Staubli VAL3: start.pgx

public program start()
begin
  // Program Rect10 start
  // Program generated by RoboDK v3.6.2 for Staubli TX200 on 17/05/2019 09:38:33
  // Using nominal kinematics.
   // mise en rotation pompe vitesse nulle
   aioSet(Tpompe,0)
   put("Tension pompe nulle")
   // arrêt pompe
   dioSet(doPompe,0)
   put("Pompe arret")

   // fermeture obturateur
   dioSet(doValve2,0)
   dioSet(doValve1,1)
   put("Obturateur fermé")
  // Afficher effecteur
  nTraj=movej(jJoint[0],tTool[0],mSpeed[0])
  nTraj=movel(pPoint[0],tTool[0],mSpeed[0])
  nTraj=movel(pPoint[1],tTool[0],mSpeed[0])
  waitEndMove()

  // ouverture obturateur
  dioSet(doValve1,0)
  dioSet(doValve2,1)
  put("Obturateur ouvert")
  delay(nTObtOpen)
  // marche pompe vitesse faible
  dioSet(doPompe,1)
  put("Pompe en marche")
  delay(nTPompeOn)
  // rotation pompe vitesse donnée
  aioSet(Tpompe,nTension)
  put("Pompe en rotation")
  nTraj=movel(pPoint[2],tTool[0],mSpeed[0])
  nTraj=movel(pPoint[3],tTool[0],mSpeed[1])
  nTraj=movel(pPoint[4],tTool[0],mSpeed[1])
  nTraj=movel(pPoint[5],tTool[0],mSpeed[1])
  nTraj=movel(pPoint[6],tTool[0],mSpeed[1])
  nTraj=movel(pPoint[7],tTool[0],mSpeed[1])
  nTraj=movel(pPoint[8],tTool[0],mSpeed[1])
  nTraj=movel(pPoint[9],tTool[0],mSpeed[1])
  nTraj=movel(pPoint[10],tTool[0],mSpeed[1])
  nTraj=movel(pPoint[11],tTool[0],mSpeed[1])
  nTraj=movel(pPoint[12],tTool[0],mSpeed[1])
  nTraj=movel(pPoint[13],tTool[0],mSpeed[1])
  nTraj=movel(pPoint[14],tTool[0],mSpeed[1])
  nTraj=movel(pPoint[15],tTool[0],mSpeed[1])
  nTraj=movel(pPoint[16],tTool[0],mSpeed[1])
  nTraj=movel(pPoint[17],tTool[0],mSpeed[1])
  nTraj=movel(pPoint[18],tTool[0],mSpeed[1])
  nTraj=movel(pPoint[19],tTool[0],mSpeed[1])
  nTraj=movel(pPoint[20],tTool[0],mSpeed[1])
  nTraj=movel(pPoint[21],tTool[0],mSpeed[1])
  nTraj=movel(pPoint[22],tTool[0],mSpeed[1])
  nTraj=movel(pPoint[23],tTool[0],mSpeed[1])
  nTraj=movel(pPoint[24],tTool[0],mSpeed[1])
  nTraj=movel(pPoint[25],tTool[0],mSpeed[1])
  nTraj=movel(pPoint[26],tTool[0],mSpeed[1])
  nTraj=movel(pPoint[27],tTool[0],mSpeed[1])
  nTraj=movel(pPoint[28],tTool[0],mSpeed[1])
  nTraj=movel(pPoint[29],tTool[0],mSpeed[1])
  nTraj=movel(pPoint[30],tTool[0],mSpeed[1])
  nTraj=movel(pPoint[31],tTool[0],mSpeed[1])
  nTraj=movel(pPoint[32],tTool[0],mSpeed[1])
  nTraj=movel(pPoint[33],tTool[0],mSpeed[1])
  nTraj=movel(pPoint[34],tTool[0],mSpeed[1])
  nTraj=movel(pPoint[35],tTool[0],mSpeed[1])
  nTraj=movel(pPoint[36],tTool[0],mSpeed[1])
  nTraj=movel(pPoint[37],tTool[0],mSpeed[1])
  nTraj=movel(pPoint[38],tTool[0],mSpeed[1])
  nTraj=movel(pPoint[39],tTool[0],mSpeed[1])
  nTraj=movel(pPoint[40],tTool[0],mSpeed[1])
  nTraj=movel(pPoint[41],tTool[0],mSpeed[1])
  nTraj=movel(pPoint[42],tTool[0],mSpeed[1])
  nTraj=movel(pPoint[43],tTool[0],mSpeed[1])
  nTraj=movel(pPoint[44],tTool[0],mSpeed[1])
  nTraj=movel(pPoint[45],tTool[0],mSpeed[1])
  nTraj=movel(pPoint[46],tTool[0],mSpeed[1])
  nTraj=movel(pPoint[47],tTool[0],mSpeed[1])
  nTraj=movel(pPoint[48],tTool[0],mSpeed[1])
  nTraj=movel(pPoint[49],tTool[0],mSpeed[1])
  nTraj=movel(pPoint[50],tTool[0],mSpeed[1])
  nTraj=movel(pPoint[51],tTool[0],mSpeed[1])
  nTraj=movel(pPoint[52],tTool[0],mSpeed[1])
  nTraj=movel(pPoint[53],tTool[0],mSpeed[1])
  nTraj=movel(pPoint[54],tTool[0],mSpeed[1])
  nTraj=movel(pPoint[55],tTool[0],mSpeed[1])
  nTraj=movel(pPoint[56],tTool[0],mSpeed[1])
  nTraj=movel(pPoint[57],tTool[0],mSpeed[1])
  nTraj=movel(pPoint[58],tTool[0],mSpeed[1])
  nTraj=movel(pPoint[59],tTool[0],mSpeed[1])
  nTraj=movel(pPoint[60],tTool[0],mSpeed[1])
  nTraj=movel(pPoint[61],tTool[0],mSpeed[1])
  nTraj=movel(pPoint[62],tTool[0],mSpeed[1])
  nTraj=movel(pPoint[63],tTool[0],mSpeed[1])
  nTraj=movel(pPoint[64],tTool[0],mSpeed[1])
  nTraj=movel(pPoint[65],tTool[0],mSpeed[1])
  nTraj=movel(pPoint[66],tTool[0],mSpeed[1])
  nTraj=movel(pPoint[67],tTool[0],mSpeed[1])
  nTraj=movel(pPoint[68],tTool[0],mSpeed[1])
  nTraj=movel(pPoint[69],tTool[0],mSpeed[1])
  nTraj=movel(pPoint[70],tTool[0],mSpeed[1])
  waitEndMove()
    // arrêt pompe
  dioSet(doPompe,0)
  put("Pompe arret")
  delay(nTPompeOff)

  // fermeture obturateur
  dioSet(doValve2,0)
  dioSet(doValve1,1)
  put("Obturateur fermé")
  nTraj=movel(pPoint[71],tTool[0],mSpeed[1])
  waitEndMove()

  nTraj=movel(pPoint[72],tTool[0],mSpeed[2])
  nTraj=movel(pPoint[73],tTool[0],mSpeed[2])
  nTraj=movel(pPoint[74],tTool[0],mSpeed[3])
  nTraj=movel(pPoint[75],tTool[0],mSpeed[3])
  waitEndMove()

  // ouverture obturateur
  dioSet(doValve1,0)
  dioSet(doValve2,1)
  put("Obturateur ouvert")
  delay(nTObtOpen)
  // marche pompe vitesse faible
  dioSet(doPompe,1)
  put("Pompe en marche")
  delay(nTPompeOn)
  // rotation pompe vitesse donnée
  aioSet(Tpompe,nTension)
  put("Pompe en rotation")
  nTraj=movel(pPoint[76],tTool[0],mSpeed[3])
  nTraj=movel(pPoint[77],tTool[0],mSpeed[4])
  nTraj=movel(pPoint[78],tTool[0],mSpeed[4])
  nTraj=movel(pPoint[79],tTool[0],mSpeed[4])
  nTraj=movel(pPoint[80],tTool[0],mSpeed[4])
  nTraj=movel(pPoint[81],tTool[0],mSpeed[4])
  nTraj=movel(pPoint[82],tTool[0],mSpeed[4])
  nTraj=movel(pPoint[83],tTool[0],mSpeed[4])
  nTraj=movel(pPoint[84],tTool[0],mSpeed[4])
  nTraj=movel(pPoint[85],tTool[0],mSpeed[4])
  nTraj=movel(pPoint[86],tTool[0],mSpeed[4])
  nTraj=movel(pPoint[87],tTool[0],mSpeed[4])
  nTraj=movel(pPoint[88],tTool[0],mSpeed[4])
  nTraj=movel(pPoint[89],tTool[0],mSpeed[4])
  nTraj=movel(pPoint[90],tTool[0],mSpeed[4])
  nTraj=movel(pPoint[91],tTool[0],mSpeed[4])
  nTraj=movel(pPoint[92],tTool[0],mSpeed[4])
  nTraj=movel(pPoint[93],tTool[0],mSpeed[4])
  nTraj=movel(pPoint[94],tTool[0],mSpeed[4])
  nTraj=movel(pPoint[95],tTool[0],mSpeed[4])
  nTraj=movel(pPoint[96],tTool[0],mSpeed[4])
  nTraj=movel(pPoint[97],tTool[0],mSpeed[4])
  nTraj=movel(pPoint[98],tTool[0],mSpeed[4])
  nTraj=movel(pPoint[99],tTool[0],mSpeed[4])
  nTraj=movel(pPoint[100],tTool[0],mSpeed[4])
  nTraj=movel(pPoint[101],tTool[0],mSpeed[4])
  nTraj=movel(pPoint[102],tTool[0],mSpeed[4])
  nTraj=movel(pPoint[103],tTool[0],mSpeed[4])
  nTraj=movel(pPoint[104],tTool[0],mSpeed[4])
  nTraj=movel(pPoint[105],tTool[0],mSpeed[4])
  nTraj=movel(pPoint[106],tTool[0],mSpeed[4])
  nTraj=movel(pPoint[107],tTool[0],mSpeed[4])
  nTraj=movel(pPoint[108],tTool[0],mSpeed[4])
  nTraj=movel(pPoint[109],tTool[0],mSpeed[4])
  nTraj=movel(pPoint[110],tTool[0],mSpeed[4])
  nTraj=movel(pPoint[111],tTool[0],mSpeed[4])
  nTraj=movel(pPoint[112],tTool[0],mSpeed[4])
  nTraj=movel(pPoint[113],tTool[0],mSpeed[4])
  nTraj=movel(pPoint[114],tTool[0],mSpeed[4])
  nTraj=movel(pPoint[115],tTool[0],mSpeed[4])
  nTraj=movel(pPoint[116],tTool[0],mSpeed[4])
  nTraj=movel(pPoint[117],tTool[0],mSpeed[4])
  nTraj=movel(pPoint[118],tTool[0],mSpeed[4])
  nTraj=movel(pPoint[119],tTool[0],mSpeed[4])
  nTraj=movel(pPoint[120],tTool[0],mSpeed[4])
  nTraj=movel(pPoint[121],tTool[0],mSpeed[4])
  nTraj=movel(pPoint[122],tTool[0],mSpeed[4])
  nTraj=movel(pPoint[123],tTool[0],mSpeed[4])
  nTraj=movel(pPoint[124],tTool[0],mSpeed[4])
  nTraj=movel(pPoint[125],tTool[0],mSpeed[4])
  nTraj=movel(pPoint[126],tTool[0],mSpeed[4])
  nTraj=movel(pPoint[127],tTool[0],mSpeed[4])
  nTraj=movel(pPoint[128],tTool[0],mSpeed[4])
  nTraj=movel(pPoint[129],tTool[0],mSpeed[4])
  nTraj=movel(pPoint[130],tTool[0],mSpeed[4])
  nTraj=movel(pPoint[131],tTool[0],mSpeed[4])
  nTraj=movel(pPoint[132],tTool[0],mSpeed[4])
  nTraj=movel(pPoint[133],tTool[0],mSpeed[4])
  nTraj=movel(pPoint[134],tTool[0],mSpeed[4])
  nTraj=movel(pPoint[135],tTool[0],mSpeed[4])
  nTraj=movel(pPoint[136],tTool[0],mSpeed[4])
  nTraj=movel(pPoint[137],tTool[0],mSpeed[4])
  nTraj=movel(pPoint[138],tTool[0],mSpeed[4])
  nTraj=movel(pPoint[139],tTool[0],mSpeed[4])
  nTraj=movel(pPoint[140],tTool[0],mSpeed[4])
  nTraj=movel(pPoint[141],tTool[0],mSpeed[4])
  nTraj=movel(pPoint[142],tTool[0],mSpeed[4])
  nTraj=movel(pPoint[143],tTool[0],mSpeed[4])
  nTraj=movel(pPoint[144],tTool[0],mSpeed[4])
    waitEndMove()

  // arrêt pompe
  dioSet(doPompe,0)
  put("Pompe arret")
  delay(nTPompeOff)

  // fermeture obturateur
  dioSet(doValve2,0)
  dioSet(doValve1,1)
  put("Obturateur fermé")
  nTraj=movel(pPoint[145],tTool[0],mSpeed[4])
  waitEndMove()

  nTraj=movel(pPoint[146],tTool[0],mSpeed[5])
  nTraj=movel(pPoint[147],tTool[0],mSpeed[5])
  nTraj=movel(pPoint[148],tTool[0],mSpeed[6])
  nTraj=movel(pPoint[149],tTool[0],mSpeed[6])
  waitEndMove()

  // ouverture obturateur
  dioSet(doValve1,0)
  dioSet(doValve2,1)
  put("Obturateur ouvert")
  delay(nTObtOpen)
  // marche pompe vitesse faible
  dioSet(doPompe,1)
  put("Pompe en marche")
  delay(nTPompeOn)
  // rotation pompe vitesse donnée
  aioSet(Tpompe,nTension)
  put("Pompe en rotation")
  nTraj=movel(pPoint[150],tTool[0],mSpeed[6])
  nTraj=movel(pPoint[151],tTool[0],mSpeed[7])
  nTraj=movel(pPoint[152],tTool[0],mSpeed[7])
  nTraj=movel(pPoint[153],tTool[0],mSpeed[7])
  nTraj=movel(pPoint[154],tTool[0],mSpeed[7])
  nTraj=movel(pPoint[155],tTool[0],mSpeed[7])
  nTraj=movel(pPoint[156],tTool[0],mSpeed[7])
  nTraj=movel(pPoint[157],tTool[0],mSpeed[7])
  nTraj=movel(pPoint[158],tTool[0],mSpeed[7])
  nTraj=movel(pPoint[159],tTool[0],mSpeed[7])
  nTraj=movel(pPoint[160],tTool[0],mSpeed[7])
  nTraj=movel(pPoint[161],tTool[0],mSpeed[7])
  nTraj=movel(pPoint[162],tTool[0],mSpeed[7])
  nTraj=movel(pPoint[163],tTool[0],mSpeed[7])
  nTraj=movel(pPoint[164],tTool[0],mSpeed[7])
  nTraj=movel(pPoint[165],tTool[0],mSpeed[7])
  nTraj=movel(pPoint[166],tTool[0],mSpeed[7])
  nTraj=movel(pPoint[167],tTool[0],mSpeed[7])
  nTraj=movel(pPoint[168],tTool[0],mSpeed[7])
  nTraj=movel(pPoint[169],tTool[0],mSpeed[7])
  nTraj=movel(pPoint[170],tTool[0],mSpeed[7])
  nTraj=movel(pPoint[171],tTool[0],mSpeed[7])
  nTraj=movel(pPoint[172],tTool[0],mSpeed[7])
  nTraj=movel(pPoint[173],tTool[0],mSpeed[7])
  nTraj=movel(pPoint[174],tTool[0],mSpeed[7])
  nTraj=movel(pPoint[175],tTool[0],mSpeed[7])
  nTraj=movel(pPoint[176],tTool[0],mSpeed[7])
  nTraj=movel(pPoint[177],tTool[0],mSpeed[7])
  nTraj=movel(pPoint[178],tTool[0],mSpeed[7])
  nTraj=movel(pPoint[179],tTool[0],mSpeed[7])
  nTraj=movel(pPoint[180],tTool[0],mSpeed[7])
  nTraj=movel(pPoint[181],tTool[0],mSpeed[7])
  nTraj=movel(pPoint[182],tTool[0],mSpeed[7])
  nTraj=movel(pPoint[183],tTool[0],mSpeed[7])
  nTraj=movel(pPoint[184],tTool[0],mSpeed[7])
  nTraj=movel(pPoint[185],tTool[0],mSpeed[7])
  nTraj=movel(pPoint[186],tTool[0],mSpeed[7])
  nTraj=movel(pPoint[187],tTool[0],mSpeed[7])
  nTraj=movel(pPoint[188],tTool[0],mSpeed[7])
  nTraj=movel(pPoint[189],tTool[0],mSpeed[7])
  nTraj=movel(pPoint[190],tTool[0],mSpeed[7])
  nTraj=movel(pPoint[191],tTool[0],mSpeed[7])
  nTraj=movel(pPoint[192],tTool[0],mSpeed[7])
  nTraj=movel(pPoint[193],tTool[0],mSpeed[7])
  nTraj=movel(pPoint[194],tTool[0],mSpeed[7])
  nTraj=movel(pPoint[195],tTool[0],mSpeed[7])
  nTraj=movel(pPoint[196],tTool[0],mSpeed[7])
  nTraj=movel(pPoint[197],tTool[0],mSpeed[7])
  nTraj=movel(pPoint[198],tTool[0],mSpeed[7])
  nTraj=movel(pPoint[199],tTool[0],mSpeed[7])
  nTraj=movel(pPoint[200],tTool[0],mSpeed[7])
  nTraj=movel(pPoint[201],tTool[0],mSpeed[7])
  nTraj=movel(pPoint[202],tTool[0],mSpeed[7])
  nTraj=movel(pPoint[203],tTool[0],mSpeed[7])
  nTraj=movel(pPoint[204],tTool[0],mSpeed[7])
  nTraj=movel(pPoint[205],tTool[0],mSpeed[7])
  nTraj=movel(pPoint[206],tTool[0],mSpeed[7])
  nTraj=movel(pPoint[207],tTool[0],mSpeed[7])
  nTraj=movel(pPoint[208],tTool[0],mSpeed[7])
  nTraj=movel(pPoint[209],tTool[0],mSpeed[7])
  nTraj=movel(pPoint[210],tTool[0],mSpeed[7])
  nTraj=movel(pPoint[211],tTool[0],mSpeed[7])
  nTraj=movel(pPoint[212],tTool[0],mSpeed[7])
  nTraj=movel(pPoint[213],tTool[0],mSpeed[7])
  nTraj=movel(pPoint[214],tTool[0],mSpeed[7])
  nTraj=movel(pPoint[215],tTool[0],mSpeed[7])
  nTraj=movel(pPoint[216],tTool[0],mSpeed[7])
  nTraj=movel(pPoint[217],tTool[0],mSpeed[7])
  nTraj=movel(pPoint[218],tTool[0],mSpeed[7])
    waitEndMove()

  // arrêt pompe
  dioSet(doPompe,0)
  put("Pompe arret")
  delay(nTPompeOff)

  // fermeture obturateur
  dioSet(doValve2,0)
  dioSet(doValve1,1)
  put("Obturateur fermé")
  nTraj=movel(pPoint[219],tTool[0],mSpeed[7])
  waitEndMove()

  nTraj=movel(pPoint[220],tTool[0],mSpeed[8])
  nTraj=movel(pPoint[221],tTool[0],mSpeed[8])
  nTraj=movel(pPoint[222],tTool[0],mSpeed[9])
  nTraj=movel(pPoint[223],tTool[0],mSpeed[9])
  waitEndMove()

  // ouverture obturateur
  dioSet(doValve1,0)
  dioSet(doValve2,1)
  put("Obturateur ouvert")
  delay(nTObtOpen)
  // marche pompe vitesse faible
  dioSet(doPompe,1)
  put("Pompe en marche")
  delay(nTPompeOn)
  // rotation pompe vitesse donnée
  aioSet(Tpompe,nTension)
  put("Pompe en rotation")
  nTraj=movel(pPoint[224],tTool[0],mSpeed[9])
  nTraj=movel(pPoint[225],tTool[0],mSpeed[10])
  nTraj=movel(pPoint[226],tTool[0],mSpeed[10])
  nTraj=movel(pPoint[227],tTool[0],mSpeed[10])
  nTraj=movel(pPoint[228],tTool[0],mSpeed[10])
  nTraj=movel(pPoint[229],tTool[0],mSpeed[10])
  nTraj=movel(pPoint[230],tTool[0],mSpeed[10])
  nTraj=movel(pPoint[231],tTool[0],mSpeed[10])
  nTraj=movel(pPoint[232],tTool[0],mSpeed[10])
  nTraj=movel(pPoint[233],tTool[0],mSpeed[10])
  nTraj=movel(pPoint[234],tTool[0],mSpeed[10])
  nTraj=movel(pPoint[235],tTool[0],mSpeed[10])
  nTraj=movel(pPoint[236],tTool[0],mSpeed[10])
  nTraj=movel(pPoint[237],tTool[0],mSpeed[10])
  nTraj=movel(pPoint[238],tTool[0],mSpeed[10])
  nTraj=movel(pPoint[239],tTool[0],mSpeed[10])
  nTraj=movel(pPoint[240],tTool[0],mSpeed[10])
  nTraj=movel(pPoint[241],tTool[0],mSpeed[10])
  nTraj=movel(pPoint[242],tTool[0],mSpeed[10])
  nTraj=movel(pPoint[243],tTool[0],mSpeed[10])
  nTraj=movel(pPoint[244],tTool[0],mSpeed[10])
  nTraj=movel(pPoint[245],tTool[0],mSpeed[10])
  nTraj=movel(pPoint[246],tTool[0],mSpeed[10])
  nTraj=movel(pPoint[247],tTool[0],mSpeed[10])
  nTraj=movel(pPoint[248],tTool[0],mSpeed[10])
  nTraj=movel(pPoint[249],tTool[0],mSpeed[10])
  nTraj=movel(pPoint[250],tTool[0],mSpeed[10])
  nTraj=movel(pPoint[251],tTool[0],mSpeed[10])
  nTraj=movel(pPoint[252],tTool[0],mSpeed[10])
  nTraj=movel(pPoint[253],tTool[0],mSpeed[10])
  nTraj=movel(pPoint[254],tTool[0],mSpeed[10])
  nTraj=movel(pPoint[255],tTool[0],mSpeed[10])
  nTraj=movel(pPoint[256],tTool[0],mSpeed[10])
  nTraj=movel(pPoint[257],tTool[0],mSpeed[10])
  nTraj=movel(pPoint[258],tTool[0],mSpeed[10])
  nTraj=movel(pPoint[259],tTool[0],mSpeed[10])
  nTraj=movel(pPoint[260],tTool[0],mSpeed[10])
  nTraj=movel(pPoint[261],tTool[0],mSpeed[10])
  nTraj=movel(pPoint[262],tTool[0],mSpeed[10])
  nTraj=movel(pPoint[263],tTool[0],mSpeed[10])
  nTraj=movel(pPoint[264],tTool[0],mSpeed[10])
  nTraj=movel(pPoint[265],tTool[0],mSpeed[10])
  nTraj=movel(pPoint[266],tTool[0],mSpeed[10])
  nTraj=movel(pPoint[267],tTool[0],mSpeed[10])
  nTraj=movel(pPoint[268],tTool[0],mSpeed[10])
  nTraj=movel(pPoint[269],tTool[0],mSpeed[10])
  nTraj=movel(pPoint[270],tTool[0],mSpeed[10])
  nTraj=movel(pPoint[271],tTool[0],mSpeed[10])
  nTraj=movel(pPoint[272],tTool[0],mSpeed[10])
  nTraj=movel(pPoint[273],tTool[0],mSpeed[10])
  nTraj=movel(pPoint[274],tTool[0],mSpeed[10])
  nTraj=movel(pPoint[275],tTool[0],mSpeed[10])
  nTraj=movel(pPoint[276],tTool[0],mSpeed[10])
  nTraj=movel(pPoint[277],tTool[0],mSpeed[10])
  nTraj=movel(pPoint[278],tTool[0],mSpeed[10])
  nTraj=movel(pPoint[279],tTool[0],mSpeed[10])
  nTraj=movel(pPoint[280],tTool[0],mSpeed[10])
  nTraj=movel(pPoint[281],tTool[0],mSpeed[10])
  nTraj=movel(pPoint[282],tTool[0],mSpeed[10])
  nTraj=movel(pPoint[283],tTool[0],mSpeed[10])
  nTraj=movel(pPoint[284],tTool[0],mSpeed[10])
  nTraj=movel(pPoint[285],tTool[0],mSpeed[10])
  nTraj=movel(pPoint[286],tTool[0],mSpeed[10])
  nTraj=movel(pPoint[287],tTool[0],mSpeed[10])
  nTraj=movel(pPoint[288],tTool[0],mSpeed[10])
  nTraj=movel(pPoint[289],tTool[0],mSpeed[10])
  nTraj=movel(pPoint[290],tTool[0],mSpeed[10])
  nTraj=movel(pPoint[291],tTool[0],mSpeed[10])
  nTraj=movel(pPoint[292],tTool[0],mSpeed[10])
    waitEndMove()

  // arrêt pompe
  dioSet(doPompe,0)
  put("Pompe arret")
  delay(nTPompeOff)

  // fermeture obturateur
  dioSet(doValve2,0)
  dioSet(doValve1,1)
  put("Obturateur fermé")
  nTraj=movel(pPoint[293],tTool[0],mSpeed[10])
  waitEndMove()


  nTraj=movel(pPoint[294],tTool[0],mSpeed[11])
  nTraj=movel(pPoint[295],tTool[0],mSpeed[11])
  nTraj=movel(pPoint[296],tTool[0],mSpeed[12])
  nTraj=movel(pPoint[297],tTool[0],mSpeed[12])
  waitEndMove()

  // ouverture obturateur
  dioSet(doValve1,0)
  dioSet(doValve2,1)
  put("Obturateur ouvert")
  delay(nTObtOpen)
  // marche pompe vitesse faible
  dioSet(doPompe,1)
  put("Pompe en marche")
  delay(nTPompeOn)
  // rotation pompe vitesse donnée
  aioSet(Tpompe,nTension)
  put("Pompe en rotation")
  nTraj=movel(pPoint[298],tTool[0],mSpeed[12])
  nTraj=movel(pPoint[299],tTool[0],mSpeed[13])
  nTraj=movel(pPoint[300],tTool[0],mSpeed[13])
  nTraj=movel(pPoint[301],tTool[0],mSpeed[13])
  nTraj=movel(pPoint[302],tTool[0],mSpeed[13])
  nTraj=movel(pPoint[303],tTool[0],mSpeed[13])
  nTraj=movel(pPoint[304],tTool[0],mSpeed[13])
  nTraj=movel(pPoint[305],tTool[0],mSpeed[13])
  nTraj=movel(pPoint[306],tTool[0],mSpeed[13])
  nTraj=movel(pPoint[307],tTool[0],mSpeed[13])
  nTraj=movel(pPoint[308],tTool[0],mSpeed[13])
  nTraj=movel(pPoint[309],tTool[0],mSpeed[13])
  nTraj=movel(pPoint[310],tTool[0],mSpeed[13])
  nTraj=movel(pPoint[311],tTool[0],mSpeed[13])
  nTraj=movel(pPoint[312],tTool[0],mSpeed[13])
  nTraj=movel(pPoint[313],tTool[0],mSpeed[13])
  nTraj=movel(pPoint[314],tTool[0],mSpeed[13])
  nTraj=movel(pPoint[315],tTool[0],mSpeed[13])
  nTraj=movel(pPoint[316],tTool[0],mSpeed[13])
  nTraj=movel(pPoint[317],tTool[0],mSpeed[13])
  nTraj=movel(pPoint[318],tTool[0],mSpeed[13])
  nTraj=movel(pPoint[319],tTool[0],mSpeed[13])
  nTraj=movel(pPoint[320],tTool[0],mSpeed[13])
  nTraj=movel(pPoint[321],tTool[0],mSpeed[13])
  nTraj=movel(pPoint[322],tTool[0],mSpeed[13])
  nTraj=movel(pPoint[323],tTool[0],mSpeed[13])
  nTraj=movel(pPoint[324],tTool[0],mSpeed[13])
  nTraj=movel(pPoint[325],tTool[0],mSpeed[13])
  nTraj=movel(pPoint[326],tTool[0],mSpeed[13])
  nTraj=movel(pPoint[327],tTool[0],mSpeed[13])
  nTraj=movel(pPoint[328],tTool[0],mSpeed[13])
  nTraj=movel(pPoint[329],tTool[0],mSpeed[13])
  nTraj=movel(pPoint[330],tTool[0],mSpeed[13])
  nTraj=movel(pPoint[331],tTool[0],mSpeed[13])
  nTraj=movel(pPoint[332],tTool[0],mSpeed[13])
  nTraj=movel(pPoint[333],tTool[0],mSpeed[13])
  nTraj=movel(pPoint[334],tTool[0],mSpeed[13])
  nTraj=movel(pPoint[335],tTool[0],mSpeed[13])
  nTraj=movel(pPoint[336],tTool[0],mSpeed[13])
  nTraj=movel(pPoint[337],tTool[0],mSpeed[13])
  nTraj=movel(pPoint[338],tTool[0],mSpeed[13])
  nTraj=movel(pPoint[339],tTool[0],mSpeed[13])
  nTraj=movel(pPoint[340],tTool[0],mSpeed[13])
  nTraj=movel(pPoint[341],tTool[0],mSpeed[13])
  nTraj=movel(pPoint[342],tTool[0],mSpeed[13])
  nTraj=movel(pPoint[343],tTool[0],mSpeed[13])
  nTraj=movel(pPoint[344],tTool[0],mSpeed[13])
  nTraj=movel(pPoint[345],tTool[0],mSpeed[13])
  nTraj=movel(pPoint[346],tTool[0],mSpeed[13])
  nTraj=movel(pPoint[347],tTool[0],mSpeed[13])
  nTraj=movel(pPoint[348],tTool[0],mSpeed[13])
  nTraj=movel(pPoint[349],tTool[0],mSpeed[13])
  nTraj=movel(pPoint[350],tTool[0],mSpeed[13])
  nTraj=movel(pPoint[351],tTool[0],mSpeed[13])
  nTraj=movel(pPoint[352],tTool[0],mSpeed[13])
  nTraj=movel(pPoint[353],tTool[0],mSpeed[13])
  nTraj=movel(pPoint[354],tTool[0],mSpeed[13])
  nTraj=movel(pPoint[355],tTool[0],mSpeed[13])
  nTraj=movel(pPoint[356],tTool[0],mSpeed[13])
  nTraj=movel(pPoint[357],tTool[0],mSpeed[13])
  nTraj=movel(pPoint[358],tTool[0],mSpeed[13])
  nTraj=movel(pPoint[359],tTool[0],mSpeed[13])
  nTraj=movel(pPoint[360],tTool[0],mSpeed[13])
  nTraj=movel(pPoint[361],tTool[0],mSpeed[13])
  nTraj=movel(pPoint[362],tTool[0],mSpeed[13])
  nTraj=movel(pPoint[363],tTool[0],mSpeed[13])
  nTraj=movel(pPoint[364],tTool[0],mSpeed[13])
  nTraj=movel(pPoint[365],tTool[0],mSpeed[13])
  nTraj=movel(pPoint[366],tTool[0],mSpeed[13])
    waitEndMove()

  // arrêt pompe
  dioSet(doPompe,0)
  put("Pompe arret")
  delay(nTPompeOff)

  // fermeture obturateur
  dioSet(doValve2,0)
  dioSet(doValve1,1)
  put("Obturateur fermé")
  nTraj=movel(pPoint[367],tTool[0],mSpeed[13])
  waitEndMove()

  nTraj=movel(pPoint[368],tTool[0],mSpeed[14])
  nTraj=movel(pPoint[369],tTool[0],mSpeed[14])
  nTraj=movel(pPoint[370],tTool[0],mSpeed[15])
  nTraj=movel(pPoint[371],tTool[0],mSpeed[15])
  waitEndMove()

  // ouverture obturateur
  dioSet(doValve1,0)
  dioSet(doValve2,1)
  put("Obturateur ouvert")
  delay(nTObtOpen)
  // marche pompe vitesse faible
  dioSet(doPompe,1)
  put("Pompe en marche")
  delay(nTPompeOn)
  // rotation pompe vitesse donnée
  aioSet(Tpompe,nTension)
  put("Pompe en rotation")
  nTraj=movel(pPoint[372],tTool[0],mSpeed[15])
  nTraj=movel(pPoint[373],tTool[0],mSpeed[16])
  nTraj=movel(pPoint[374],tTool[0],mSpeed[16])
  nTraj=movel(pPoint[375],tTool[0],mSpeed[16])
  nTraj=movel(pPoint[376],tTool[0],mSpeed[16])
  nTraj=movel(pPoint[377],tTool[0],mSpeed[16])
  nTraj=movel(pPoint[378],tTool[0],mSpeed[16])
  nTraj=movel(pPoint[379],tTool[0],mSpeed[16])
  nTraj=movel(pPoint[380],tTool[0],mSpeed[16])
  nTraj=movel(pPoint[381],tTool[0],mSpeed[16])
  nTraj=movel(pPoint[382],tTool[0],mSpeed[16])
  nTraj=movel(pPoint[383],tTool[0],mSpeed[16])
  nTraj=movel(pPoint[384],tTool[0],mSpeed[16])
  nTraj=movel(pPoint[385],tTool[0],mSpeed[16])
  nTraj=movel(pPoint[386],tTool[0],mSpeed[16])
  nTraj=movel(pPoint[387],tTool[0],mSpeed[16])
  nTraj=movel(pPoint[388],tTool[0],mSpeed[16])
  nTraj=movel(pPoint[389],tTool[0],mSpeed[16])
  nTraj=movel(pPoint[390],tTool[0],mSpeed[16])
  nTraj=movel(pPoint[391],tTool[0],mSpeed[16])
  nTraj=movel(pPoint[392],tTool[0],mSpeed[16])
  nTraj=movel(pPoint[393],tTool[0],mSpeed[16])
  nTraj=movel(pPoint[394],tTool[0],mSpeed[16])
  nTraj=movel(pPoint[395],tTool[0],mSpeed[16])
  nTraj=movel(pPoint[396],tTool[0],mSpeed[16])
  nTraj=movel(pPoint[397],tTool[0],mSpeed[16])
  nTraj=movel(pPoint[398],tTool[0],mSpeed[16])
  nTraj=movel(pPoint[399],tTool[0],mSpeed[16])
  nTraj=movel(pPoint[400],tTool[0],mSpeed[16])
  nTraj=movel(pPoint[401],tTool[0],mSpeed[16])
  nTraj=movel(pPoint[402],tTool[0],mSpeed[16])
  nTraj=movel(pPoint[403],tTool[0],mSpeed[16])
  nTraj=movel(pPoint[404],tTool[0],mSpeed[16])
  nTraj=movel(pPoint[405],tTool[0],mSpeed[16])
  nTraj=movel(pPoint[406],tTool[0],mSpeed[16])
  nTraj=movel(pPoint[407],tTool[0],mSpeed[16])
  nTraj=movel(pPoint[408],tTool[0],mSpeed[16])
  nTraj=movel(pPoint[409],tTool[0],mSpeed[16])
  nTraj=movel(pPoint[410],tTool[0],mSpeed[16])
  nTraj=movel(pPoint[411],tTool[0],mSpeed[16])
  nTraj=movel(pPoint[412],tTool[0],mSpeed[16])
  nTraj=movel(pPoint[413],tTool[0],mSpeed[16])
  nTraj=movel(pPoint[414],tTool[0],mSpeed[16])
  nTraj=movel(pPoint[415],tTool[0],mSpeed[16])
  nTraj=movel(pPoint[416],tTool[0],mSpeed[16])
  nTraj=movel(pPoint[417],tTool[0],mSpeed[16])
  nTraj=movel(pPoint[418],tTool[0],mSpeed[16])
  nTraj=movel(pPoint[419],tTool[0],mSpeed[16])
  nTraj=movel(pPoint[420],tTool[0],mSpeed[16])
  nTraj=movel(pPoint[421],tTool[0],mSpeed[16])
  nTraj=movel(pPoint[422],tTool[0],mSpeed[16])
  nTraj=movel(pPoint[423],tTool[0],mSpeed[16])
  nTraj=movel(pPoint[424],tTool[0],mSpeed[16])
  nTraj=movel(pPoint[425],tTool[0],mSpeed[16])
  nTraj=movel(pPoint[426],tTool[0],mSpeed[16])
  nTraj=movel(pPoint[427],tTool[0],mSpeed[16])
  nTraj=movel(pPoint[428],tTool[0],mSpeed[16])
  nTraj=movel(pPoint[429],tTool[0],mSpeed[16])
  nTraj=movel(pPoint[430],tTool[0],mSpeed[16])
  nTraj=movel(pPoint[431],tTool[0],mSpeed[16])
  nTraj=movel(pPoint[432],tTool[0],mSpeed[16])
  nTraj=movel(pPoint[433],tTool[0],mSpeed[16])
  nTraj=movel(pPoint[434],tTool[0],mSpeed[16])
  nTraj=movel(pPoint[435],tTool[0],mSpeed[16])
  nTraj=movel(pPoint[436],tTool[0],mSpeed[16])
  nTraj=movel(pPoint[437],tTool[0],mSpeed[16])
  nTraj=movel(pPoint[438],tTool[0],mSpeed[16])
  nTraj=movel(pPoint[439],tTool[0],mSpeed[16])
  nTraj=movel(pPoint[440],tTool[0],mSpeed[16])
    waitEndMove()

  // arrêt pompe
  dioSet(doPompe,0)
  put("Pompe arret")
  delay(nTPompeOff)

  // fermeture obturateur
  dioSet(doValve2,0)
  dioSet(doValve1,1)
  put("Obturateur fermé")
  nTraj=movel(pPoint[441],tTool[0],mSpeed[16])
  waitEndMove()

  nTraj=movel(pPoint[442],tTool[0],mSpeed[17])
  nTraj=movel(pPoint[443],tTool[0],mSpeed[17])
  nTraj=movel(pPoint[444],tTool[0],mSpeed[18])
  nTraj=movel(pPoint[445],tTool[0],mSpeed[18])
  waitEndMove()

  // ouverture obturateur
  dioSet(doValve1,0)
  dioSet(doValve2,1)
  put("Obturateur ouvert")
  delay(nTObtOpen)
  // marche pompe vitesse faible
  dioSet(doPompe,1)
  put("Pompe en marche")
  delay(nTPompeOn)
  // rotation pompe vitesse donnée
  aioSet(Tpompe,nTension)
  put("Pompe en rotation")
  nTraj=movel(pPoint[446],tTool[0],mSpeed[18])
  nTraj=movel(pPoint[447],tTool[0],mSpeed[19])
  nTraj=movel(pPoint[448],tTool[0],mSpeed[19])
  nTraj=movel(pPoint[449],tTool[0],mSpeed[19])
  nTraj=movel(pPoint[450],tTool[0],mSpeed[19])
  nTraj=movel(pPoint[451],tTool[0],mSpeed[19])
  nTraj=movel(pPoint[452],tTool[0],mSpeed[19])
  nTraj=movel(pPoint[453],tTool[0],mSpeed[19])
  nTraj=movel(pPoint[454],tTool[0],mSpeed[19])
  nTraj=movel(pPoint[455],tTool[0],mSpeed[19])
  nTraj=movel(pPoint[456],tTool[0],mSpeed[19])
  nTraj=movel(pPoint[457],tTool[0],mSpeed[19])
  nTraj=movel(pPoint[458],tTool[0],mSpeed[19])
  nTraj=movel(pPoint[459],tTool[0],mSpeed[19])
  nTraj=movel(pPoint[460],tTool[0],mSpeed[19])
  nTraj=movel(pPoint[461],tTool[0],mSpeed[19])
  nTraj=movel(pPoint[462],tTool[0],mSpeed[19])
  nTraj=movel(pPoint[463],tTool[0],mSpeed[19])
  nTraj=movel(pPoint[464],tTool[0],mSpeed[19])
  nTraj=movel(pPoint[465],tTool[0],mSpeed[19])
  nTraj=movel(pPoint[466],tTool[0],mSpeed[19])
  nTraj=movel(pPoint[467],tTool[0],mSpeed[19])
  nTraj=movel(pPoint[468],tTool[0],mSpeed[19])
  nTraj=movel(pPoint[469],tTool[0],mSpeed[19])
  nTraj=movel(pPoint[470],tTool[0],mSpeed[19])
  nTraj=movel(pPoint[471],tTool[0],mSpeed[19])
  nTraj=movel(pPoint[472],tTool[0],mSpeed[19])
  nTraj=movel(pPoint[473],tTool[0],mSpeed[19])
  nTraj=movel(pPoint[474],tTool[0],mSpeed[19])
  nTraj=movel(pPoint[475],tTool[0],mSpeed[19])
  nTraj=movel(pPoint[476],tTool[0],mSpeed[19])
  nTraj=movel(pPoint[477],tTool[0],mSpeed[19])
  nTraj=movel(pPoint[478],tTool[0],mSpeed[19])
  nTraj=movel(pPoint[479],tTool[0],mSpeed[19])
  nTraj=movel(pPoint[480],tTool[0],mSpeed[19])
  nTraj=movel(pPoint[481],tTool[0],mSpeed[19])
  nTraj=movel(pPoint[482],tTool[0],mSpeed[19])
  nTraj=movel(pPoint[483],tTool[0],mSpeed[19])
  nTraj=movel(pPoint[484],tTool[0],mSpeed[19])
  nTraj=movel(pPoint[485],tTool[0],mSpeed[19])
  nTraj=movel(pPoint[486],tTool[0],mSpeed[19])
  nTraj=movel(pPoint[487],tTool[0],mSpeed[19])
  nTraj=movel(pPoint[488],tTool[0],mSpeed[19])
  nTraj=movel(pPoint[489],tTool[0],mSpeed[19])
  nTraj=movel(pPoint[490],tTool[0],mSpeed[19])
  nTraj=movel(pPoint[491],tTool[0],mSpeed[19])
  nTraj=movel(pPoint[492],tTool[0],mSpeed[19])
  nTraj=movel(pPoint[493],tTool[0],mSpeed[19])
  nTraj=movel(pPoint[494],tTool[0],mSpeed[19])
  nTraj=movel(pPoint[495],tTool[0],mSpeed[19])
  nTraj=movel(pPoint[496],tTool[0],mSpeed[19])
  nTraj=movel(pPoint[497],tTool[0],mSpeed[19])
  nTraj=movel(pPoint[498],tTool[0],mSpeed[19])
  nTraj=movel(pPoint[499],tTool[0],mSpeed[19])
  nTraj=movel(pPoint[500],tTool[0],mSpeed[19])
  nTraj=movel(pPoint[501],tTool[0],mSpeed[19])
  nTraj=movel(pPoint[502],tTool[0],mSpeed[19])
  nTraj=movel(pPoint[503],tTool[0],mSpeed[19])
  nTraj=movel(pPoint[504],tTool[0],mSpeed[19])
  nTraj=movel(pPoint[505],tTool[0],mSpeed[19])
  nTraj=movel(pPoint[506],tTool[0],mSpeed[19])
  nTraj=movel(pPoint[507],tTool[0],mSpeed[19])
  nTraj=movel(pPoint[508],tTool[0],mSpeed[19])
  nTraj=movel(pPoint[509],tTool[0],mSpeed[19])
  nTraj=movel(pPoint[510],tTool[0],mSpeed[19])
  nTraj=movel(pPoint[511],tTool[0],mSpeed[19])
  nTraj=movel(pPoint[512],tTool[0],mSpeed[19])
  nTraj=movel(pPoint[513],tTool[0],mSpeed[19])
  nTraj=movel(pPoint[514],tTool[0],mSpeed[19])
    waitEndMove()

  // arrêt pompe
  dioSet(doPompe,0)
  put("Pompe arret")
  delay(nTPompeOff)

  // fermeture obturateur
  dioSet(doValve2,0)
  dioSet(doValve1,1)
  put("Obturateur fermé")
  nTraj=movel(pPoint[515],tTool[0],mSpeed[19])
  waitEndMove()

  nTraj=movel(pPoint[516],tTool[0],mSpeed[20])
  nTraj=movel(pPoint[517],tTool[0],mSpeed[20])
  nTraj=movel(pPoint[518],tTool[0],mSpeed[21])
  nTraj=movel(pPoint[519],tTool[0],mSpeed[21])
  waitEndMove()

  // ouverture obturateur
  dioSet(doValve1,0)
  dioSet(doValve2,1)
  put("Obturateur ouvert")
  delay(nTObtOpen)
  // marche pompe vitesse faible
  dioSet(doPompe,1)
  put("Pompe en marche")
  delay(nTPompeOn)
  // rotation pompe vitesse donnée
  aioSet(Tpompe,nTension)
  put("Pompe en rotation")
  nTraj=movel(pPoint[520],tTool[0],mSpeed[21])
  nTraj=movel(pPoint[521],tTool[0],mSpeed[22])
  nTraj=movel(pPoint[522],tTool[0],mSpeed[22])
  nTraj=movel(pPoint[523],tTool[0],mSpeed[22])
  nTraj=movel(pPoint[524],tTool[0],mSpeed[22])
  nTraj=movel(pPoint[525],tTool[0],mSpeed[22])
  nTraj=movel(pPoint[526],tTool[0],mSpeed[22])
  nTraj=movel(pPoint[527],tTool[0],mSpeed[22])
  nTraj=movel(pPoint[528],tTool[0],mSpeed[22])
  nTraj=movel(pPoint[529],tTool[0],mSpeed[22])
  nTraj=movel(pPoint[530],tTool[0],mSpeed[22])
  nTraj=movel(pPoint[531],tTool[0],mSpeed[22])
  nTraj=movel(pPoint[532],tTool[0],mSpeed[22])
  nTraj=movel(pPoint[533],tTool[0],mSpeed[22])
  nTraj=movel(pPoint[534],tTool[0],mSpeed[22])
  nTraj=movel(pPoint[535],tTool[0],mSpeed[22])
  nTraj=movel(pPoint[536],tTool[0],mSpeed[22])
  nTraj=movel(pPoint[537],tTool[0],mSpeed[22])
  nTraj=movel(pPoint[538],tTool[0],mSpeed[22])
  nTraj=movel(pPoint[539],tTool[0],mSpeed[22])
  nTraj=movel(pPoint[540],tTool[0],mSpeed[22])
  nTraj=movel(pPoint[541],tTool[0],mSpeed[22])
  nTraj=movel(pPoint[542],tTool[0],mSpeed[22])
  nTraj=movel(pPoint[543],tTool[0],mSpeed[22])
  nTraj=movel(pPoint[544],tTool[0],mSpeed[22])
  nTraj=movel(pPoint[545],tTool[0],mSpeed[22])
  nTraj=movel(pPoint[546],tTool[0],mSpeed[22])
  nTraj=movel(pPoint[547],tTool[0],mSpeed[22])
  nTraj=movel(pPoint[548],tTool[0],mSpeed[22])
  nTraj=movel(pPoint[549],tTool[0],mSpeed[22])
  nTraj=movel(pPoint[550],tTool[0],mSpeed[22])
  nTraj=movel(pPoint[551],tTool[0],mSpeed[22])
  nTraj=movel(pPoint[552],tTool[0],mSpeed[22])
  nTraj=movel(pPoint[553],tTool[0],mSpeed[22])
  nTraj=movel(pPoint[554],tTool[0],mSpeed[22])
  nTraj=movel(pPoint[555],tTool[0],mSpeed[22])
  nTraj=movel(pPoint[556],tTool[0],mSpeed[22])
  nTraj=movel(pPoint[557],tTool[0],mSpeed[22])
  nTraj=movel(pPoint[558],tTool[0],mSpeed[22])
  nTraj=movel(pPoint[559],tTool[0],mSpeed[22])
  nTraj=movel(pPoint[560],tTool[0],mSpeed[22])
  nTraj=movel(pPoint[561],tTool[0],mSpeed[22])
  nTraj=movel(pPoint[562],tTool[0],mSpeed[22])
  nTraj=movel(pPoint[563],tTool[0],mSpeed[22])
  nTraj=movel(pPoint[564],tTool[0],mSpeed[22])
  nTraj=movel(pPoint[565],tTool[0],mSpeed[22])
  nTraj=movel(pPoint[566],tTool[0],mSpeed[22])
  nTraj=movel(pPoint[567],tTool[0],mSpeed[22])
  nTraj=movel(pPoint[568],tTool[0],mSpeed[22])
  nTraj=movel(pPoint[569],tTool[0],mSpeed[22])
  nTraj=movel(pPoint[570],tTool[0],mSpeed[22])
  nTraj=movel(pPoint[571],tTool[0],mSpeed[22])
  nTraj=movel(pPoint[572],tTool[0],mSpeed[22])
  nTraj=movel(pPoint[573],tTool[0],mSpeed[22])
  nTraj=movel(pPoint[574],tTool[0],mSpeed[22])
  nTraj=movel(pPoint[575],tTool[0],mSpeed[22])
  nTraj=movel(pPoint[576],tTool[0],mSpeed[22])
  nTraj=movel(pPoint[577],tTool[0],mSpeed[22])
  nTraj=movel(pPoint[578],tTool[0],mSpeed[22])
  nTraj=movel(pPoint[579],tTool[0],mSpeed[22])
  nTraj=movel(pPoint[580],tTool[0],mSpeed[22])
  nTraj=movel(pPoint[581],tTool[0],mSpeed[22])
  nTraj=movel(pPoint[582],tTool[0],mSpeed[22])
  nTraj=movel(pPoint[583],tTool[0],mSpeed[22])
  nTraj=movel(pPoint[584],tTool[0],mSpeed[22])
  nTraj=movel(pPoint[585],tTool[0],mSpeed[22])
  nTraj=movel(pPoint[586],tTool[0],mSpeed[22])
  nTraj=movel(pPoint[587],tTool[0],mSpeed[22])
  nTraj=movel(pPoint[588],tTool[0],mSpeed[22])
    waitEndMove()

  // arrêt pompe
  dioSet(doPompe,0)
  put("Pompe arret")
  delay(nTPompeOff)

  // fermeture obturateur
  dioSet(doValve2,0)
  dioSet(doValve1,1)
  put("Obturateur fermé")
  nTraj=movel(pPoint[589],tTool[0],mSpeed[22])
  waitEndMove()

  nTraj=movel(pPoint[590],tTool[0],mSpeed[23])
  nTraj=movel(pPoint[591],tTool[0],mSpeed[23])
  nTraj=movel(pPoint[592],tTool[0],mSpeed[24])
  nTraj=movel(pPoint[593],tTool[0],mSpeed[24])
  waitEndMove()

  // ouverture obturateur
  dioSet(doValve1,0)
  dioSet(doValve2,1)
  put("Obturateur ouvert")
  delay(nTObtOpen)
  // marche pompe vitesse faible
  dioSet(doPompe,1)
  put("Pompe en marche")
  delay(nTPompeOn)
  // rotation pompe vitesse donnée
  aioSet(Tpompe,nTension)
  put("Pompe en rotation")
  nTraj=movel(pPoint[594],tTool[0],mSpeed[24])
  nTraj=movel(pPoint[595],tTool[0],mSpeed[25])
  nTraj=movel(pPoint[596],tTool[0],mSpeed[25])
  nTraj=movel(pPoint[597],tTool[0],mSpeed[25])
  nTraj=movel(pPoint[598],tTool[0],mSpeed[25])
  nTraj=movel(pPoint[599],tTool[0],mSpeed[25])
  nTraj=movel(pPoint[600],tTool[0],mSpeed[25])
  nTraj=movel(pPoint[601],tTool[0],mSpeed[25])
  nTraj=movel(pPoint[602],tTool[0],mSpeed[25])
  nTraj=movel(pPoint[603],tTool[0],mSpeed[25])
  nTraj=movel(pPoint[604],tTool[0],mSpeed[25])
  nTraj=movel(pPoint[605],tTool[0],mSpeed[25])
  nTraj=movel(pPoint[606],tTool[0],mSpeed[25])
  nTraj=movel(pPoint[607],tTool[0],mSpeed[25])
  nTraj=movel(pPoint[608],tTool[0],mSpeed[25])
  nTraj=movel(pPoint[609],tTool[0],mSpeed[25])
  nTraj=movel(pPoint[610],tTool[0],mSpeed[25])
  nTraj=movel(pPoint[611],tTool[0],mSpeed[25])
  nTraj=movel(pPoint[612],tTool[0],mSpeed[25])
  nTraj=movel(pPoint[613],tTool[0],mSpeed[25])
  nTraj=movel(pPoint[614],tTool[0],mSpeed[25])
  nTraj=movel(pPoint[615],tTool[0],mSpeed[25])
  nTraj=movel(pPoint[616],tTool[0],mSpeed[25])
  nTraj=movel(pPoint[617],tTool[0],mSpeed[25])
  nTraj=movel(pPoint[618],tTool[0],mSpeed[25])
  nTraj=movel(pPoint[619],tTool[0],mSpeed[25])
  nTraj=movel(pPoint[620],tTool[0],mSpeed[25])
  nTraj=movel(pPoint[621],tTool[0],mSpeed[25])
  nTraj=movel(pPoint[622],tTool[0],mSpeed[25])
  nTraj=movel(pPoint[623],tTool[0],mSpeed[25])
  nTraj=movel(pPoint[624],tTool[0],mSpeed[25])
  nTraj=movel(pPoint[625],tTool[0],mSpeed[25])
  nTraj=movel(pPoint[626],tTool[0],mSpeed[25])
  nTraj=movel(pPoint[627],tTool[0],mSpeed[25])
  nTraj=movel(pPoint[628],tTool[0],mSpeed[25])
  nTraj=movel(pPoint[629],tTool[0],mSpeed[25])
  nTraj=movel(pPoint[630],tTool[0],mSpeed[25])
  nTraj=movel(pPoint[631],tTool[0],mSpeed[25])
  nTraj=movel(pPoint[632],tTool[0],mSpeed[25])
  nTraj=movel(pPoint[633],tTool[0],mSpeed[25])
  nTraj=movel(pPoint[634],tTool[0],mSpeed[25])
  nTraj=movel(pPoint[635],tTool[0],mSpeed[25])
  nTraj=movel(pPoint[636],tTool[0],mSpeed[25])
  nTraj=movel(pPoint[637],tTool[0],mSpeed[25])
  nTraj=movel(pPoint[638],tTool[0],mSpeed[25])
  nTraj=movel(pPoint[639],tTool[0],mSpeed[25])
  nTraj=movel(pPoint[640],tTool[0],mSpeed[25])
  nTraj=movel(pPoint[641],tTool[0],mSpeed[25])
  nTraj=movel(pPoint[642],tTool[0],mSpeed[25])
  nTraj=movel(pPoint[643],tTool[0],mSpeed[25])
  nTraj=movel(pPoint[644],tTool[0],mSpeed[25])
  nTraj=movel(pPoint[645],tTool[0],mSpeed[25])
  nTraj=movel(pPoint[646],tTool[0],mSpeed[25])
  nTraj=movel(pPoint[647],tTool[0],mSpeed[25])
  nTraj=movel(pPoint[648],tTool[0],mSpeed[25])
  nTraj=movel(pPoint[649],tTool[0],mSpeed[25])
  nTraj=movel(pPoint[650],tTool[0],mSpeed[25])
  nTraj=movel(pPoint[651],tTool[0],mSpeed[25])
  nTraj=movel(pPoint[652],tTool[0],mSpeed[25])
  nTraj=movel(pPoint[653],tTool[0],mSpeed[25])
  nTraj=movel(pPoint[654],tTool[0],mSpeed[25])
  nTraj=movel(pPoint[655],tTool[0],mSpeed[25])
  nTraj=movel(pPoint[656],tTool[0],mSpeed[25])
  nTraj=movel(pPoint[657],tTool[0],mSpeed[25])
  nTraj=movel(pPoint[658],tTool[0],mSpeed[25])
  nTraj=movel(pPoint[659],tTool[0],mSpeed[25])
  nTraj=movel(pPoint[660],tTool[0],mSpeed[25])
  nTraj=movel(pPoint[661],tTool[0],mSpeed[25])
  nTraj=movel(pPoint[662],tTool[0],mSpeed[25])
    waitEndMove()

  // arrêt pompe
  dioSet(doPompe,0)
  put("Pompe arret")
  delay(nTPompeOff)

  // fermeture obturateur
  dioSet(doValve2,0)
  dioSet(doValve1,1)
  put("Obturateur fermé")
  nTraj=movel(pPoint[663],tTool[0],mSpeed[25])
  waitEndMove()

  nTraj=movel(pPoint[664],tTool[0],mSpeed[26])
  nTraj=movel(pPoint[665],tTool[0],mSpeed[26])
  nTraj=movel(pPoint[666],tTool[0],mSpeed[27])
  nTraj=movel(pPoint[667],tTool[0],mSpeed[27])
  waitEndMove()

  // ouverture obturateur
  dioSet(doValve1,0)
  dioSet(doValve2,1)
  put("Obturateur ouvert")
  delay(nTObtOpen)
  // marche pompe vitesse faible
  dioSet(doPompe,1)
  put("Pompe en marche")
  delay(nTPompeOn)
  // rotation pompe vitesse donnée
  aioSet(Tpompe,nTension)
  put("Pompe en rotation")
  nTraj=movel(pPoint[668],tTool[0],mSpeed[27])
  nTraj=movel(pPoint[669],tTool[0],mSpeed[28])
  nTraj=movel(pPoint[670],tTool[0],mSpeed[28])
  nTraj=movel(pPoint[671],tTool[0],mSpeed[28])
  nTraj=movel(pPoint[672],tTool[0],mSpeed[28])
  nTraj=movel(pPoint[673],tTool[0],mSpeed[28])
  nTraj=movel(pPoint[674],tTool[0],mSpeed[28])
  nTraj=movel(pPoint[675],tTool[0],mSpeed[28])
  nTraj=movel(pPoint[676],tTool[0],mSpeed[28])
  nTraj=movel(pPoint[677],tTool[0],mSpeed[28])
  nTraj=movel(pPoint[678],tTool[0],mSpeed[28])
  nTraj=movel(pPoint[679],tTool[0],mSpeed[28])
  nTraj=movel(pPoint[680],tTool[0],mSpeed[28])
  nTraj=movel(pPoint[681],tTool[0],mSpeed[28])
  nTraj=movel(pPoint[682],tTool[0],mSpeed[28])
  nTraj=movel(pPoint[683],tTool[0],mSpeed[28])
  nTraj=movel(pPoint[684],tTool[0],mSpeed[28])
  nTraj=movel(pPoint[685],tTool[0],mSpeed[28])
  nTraj=movel(pPoint[686],tTool[0],mSpeed[28])
  nTraj=movel(pPoint[687],tTool[0],mSpeed[28])
  nTraj=movel(pPoint[688],tTool[0],mSpeed[28])
  nTraj=movel(pPoint[689],tTool[0],mSpeed[28])
  nTraj=movel(pPoint[690],tTool[0],mSpeed[28])
  nTraj=movel(pPoint[691],tTool[0],mSpeed[28])
  nTraj=movel(pPoint[692],tTool[0],mSpeed[28])
  nTraj=movel(pPoint[693],tTool[0],mSpeed[28])
  nTraj=movel(pPoint[694],tTool[0],mSpeed[28])
  nTraj=movel(pPoint[695],tTool[0],mSpeed[28])
  nTraj=movel(pPoint[696],tTool[0],mSpeed[28])
  nTraj=movel(pPoint[697],tTool[0],mSpeed[28])
  nTraj=movel(pPoint[698],tTool[0],mSpeed[28])
  nTraj=movel(pPoint[699],tTool[0],mSpeed[28])
  nTraj=movel(pPoint[700],tTool[0],mSpeed[28])
  nTraj=movel(pPoint[701],tTool[0],mSpeed[28])
  nTraj=movel(pPoint[702],tTool[0],mSpeed[28])
  nTraj=movel(pPoint[703],tTool[0],mSpeed[28])
  nTraj=movel(pPoint[704],tTool[0],mSpeed[28])
  nTraj=movel(pPoint[705],tTool[0],mSpeed[28])
  nTraj=movel(pPoint[706],tTool[0],mSpeed[28])
  nTraj=movel(pPoint[707],tTool[0],mSpeed[28])
  nTraj=movel(pPoint[708],tTool[0],mSpeed[28])
  nTraj=movel(pPoint[709],tTool[0],mSpeed[28])
  nTraj=movel(pPoint[710],tTool[0],mSpeed[28])
  nTraj=movel(pPoint[711],tTool[0],mSpeed[28])
  nTraj=movel(pPoint[712],tTool[0],mSpeed[28])
  nTraj=movel(pPoint[713],tTool[0],mSpeed[28])
  nTraj=movel(pPoint[714],tTool[0],mSpeed[28])
  nTraj=movel(pPoint[715],tTool[0],mSpeed[28])
  nTraj=movel(pPoint[716],tTool[0],mSpeed[28])
  nTraj=movel(pPoint[717],tTool[0],mSpeed[28])
  nTraj=movel(pPoint[718],tTool[0],mSpeed[28])
  nTraj=movel(pPoint[719],tTool[0],mSpeed[28])
  nTraj=movel(pPoint[720],tTool[0],mSpeed[28])
  nTraj=movel(pPoint[721],tTool[0],mSpeed[28])
  nTraj=movel(pPoint[722],tTool[0],mSpeed[28])
  nTraj=movel(pPoint[723],tTool[0],mSpeed[28])
  nTraj=movel(pPoint[724],tTool[0],mSpeed[28])
  nTraj=movel(pPoint[725],tTool[0],mSpeed[28])
  nTraj=movel(pPoint[726],tTool[0],mSpeed[28])
  nTraj=movel(pPoint[727],tTool[0],mSpeed[28])
  nTraj=movel(pPoint[728],tTool[0],mSpeed[28])
  nTraj=movel(pPoint[729],tTool[0],mSpeed[28])
  nTraj=movel(pPoint[730],tTool[0],mSpeed[28])
  nTraj=movel(pPoint[731],tTool[0],mSpeed[28])
  nTraj=movel(pPoint[732],tTool[0],mSpeed[28])
  nTraj=movel(pPoint[733],tTool[0],mSpeed[28])
  nTraj=movel(pPoint[734],tTool[0],mSpeed[28])
  nTraj=movel(pPoint[735],tTool[0],mSpeed[28])
  nTraj=movel(pPoint[736],tTool[0],mSpeed[28])
  nTraj=movel(pPoint[737],tTool[0],mSpeed[28])
  waitEndMove()

  // arrêt pompe
  dioSet(doPompe,0)
  put("Pompe arret")
  delay(nTPompeOff)

  // fermeture obturateur
  dioSet(doValve2,0)
  dioSet(doValve1,1)
  put("Obturateur fermé")
  nTraj=movel(pPoint[738],tTool[0],mSpeed[29])
  nTraj=movel(pPoint[739],tTool[0],mSpeed[29])

  waitEndMove()
  // Program Rect10 end

end
